FUNCTION_BLOCK FB_CheckMaterial_SFC
VAR_INPUT
	// SFC-Flags
    SFCPause: BOOL;
    SFCReset: BOOL;
    
    // Indicadores de sincronizacion
    Ack: BOOL := TRUE;
    Execute: BOOL;
	
	//Entradas
	Base_en_Alimentador: BOOL;
	Pulsador_marcha: BOOL;
END_VAR
VAR_OUTPUT
	// Indicadores de sincronizacion
    Done: BOOL;
    Ready: BOOL;
	
	//Salidas
	LamparaAlarma: BOOL;
	Lampara_falta_material: BOOL;
END_VAR
VAR
	TMAt: TIME := T#1S;
END_VAR

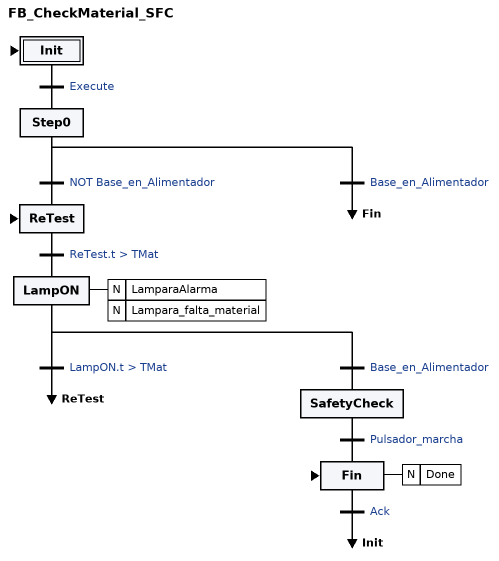
INITIAL_STEP Init:
END_STEP
TRANSITION FROM Init TO Step0
    := Execute;
END_TRANSITION
STEP Step0:
END_STEP
TRANSITION FROM Step0 TO ReTest
    := NOT Base_en_Alimentador;
END_TRANSITION
STEP ReTest:
END_STEP
TRANSITION FROM ReTest TO LampON
    := ReTest.t > TMat;
END_TRANSITION
TRANSITION FROM Step0 TO Fin
    := Base_en_Alimentador;
END_TRANSITION
STEP LampON:
    LamparaAlarma(N);
    Lampara_falta_material(N);
END_STEP
TRANSITION FROM LampON TO ReTest
    := LampON.t > TMat;
END_TRANSITION
TRANSITION FROM LampON TO SafetyCheck
    := Base_en_Alimentador;
END_TRANSITION
STEP SafetyCheck:
END_STEP
TRANSITION FROM SafetyCheck TO Fin
    := Pulsador_marcha;
END_TRANSITION
STEP Fin:
    Done(N);
END_STEP
TRANSITION FROM Fin TO Init
    := Ack;
END_TRANSITION

END_FUNCTION_BLOCK

(* stored: Version 1.1.0.1, ProductVersion 3.1.4024.12
   POU FB_CheckMaterial_SFC: Id {3af8f292-ab0d-4949-849c-a31fe1741044}, SpecialFunc None *)
